FUNCTION_BLOCK FB_UpperLimitRetrieval
VAR_INPUT
    bStartDCA : BOOL;
    bUpdateRequested : BOOL;
    fTfruitHot : REAL; // fruit temperature at hot side of the room
    fTfruitCold : REAL; // fruit temperature at cold side of the room
END_VAR
VAR_OUTPUT
    fLatestUpperLimit : REAL ;
	fCurrentUpperLimit : REAL := 999.99; //If fCurrentUpperLimit = 999.99 then we know that it isn't set yet
END_VAR
VAR
	bDcaStarted : BOOL := FALSE;
    fStartDiff_upperlimit : REAL;
    fEndDiff_upperlimit : REAL;
    fMax_upperlimit : REAL;
    tTimeForUpperLimitLog : TIME := T#30M;
    bTimer_done : BOOL;
	timer : TON;
END_VAR

R_trig(CLK:=bStartDCA);
IF R_trig.Q THEN // positive edge trigger of a DCA action
	bDcaStarted:= TRUE;
END_IF

IF bDcaStarted THEN
    fStartDiff_upperlimit := ABS(fTfruitHot - fTfruitCold);
    timer(IN := bDcaStarted, PT := tTimeForUpperLimitLog, Q => bTimer_done); // wait for 20 minutes
    IF bTimer_done THEN
        fEndDiff_upperlimit := ABS(fTfruitHot - fTfruitCold);
        fMax_upperlimit := fStartDiff_upperlimit - fEndDiff_upperlimit;
        fLatestUpperLimit := fMax_upperlimit;
		bDcaStarted := FALSE;
    END_IF
END_IF

IF bUpdateRequested THEN
    fCurrentUpperLimit := fLatestUpperLimit;
END_IF

END_FUNCTION_BLOCK

(* stored: Version 1.1.0.1, ProductVersion 3.1.4024.11
   POU FB_UpperLimitRetrieval: Id {d3c41b8e-58ad-4411-aa53-da5f8e9961d0}, SpecialFunc None *)
